(* Logix 5000 project; controller WWTP_SEC_CLX vendor 1 type 14 code 54 rev 17.2; software revision 17.00; part 12 of 13 *)
(* tags used below, declared in another part *)
   I_M403_Fault : ALIAS FOR Local:3:I.DATA.4;
   I_M403_Fault_IOFault : ALIAS FOR Local:3:I.Fault.4;
   I_M403_InAuto : ALIAS FOR Local:3:I.DATA.5;
   I_M403_InAuto_IOFault : ALIAS FOR Local:3:I.Fault.5;
   I_M403_RunFdbk : ALIAS FOR Local:3:I.DATA.3;
   I_M403_RunFdbk_IOFault : ALIAS FOR Local:3:I.Fault.3;
   I_SecTk01_InAuto : ALIAS FOR Local:2:I.DATA.4;
   I_SecTk01_InAuto_IOFault : ALIAS FOR Local:2:I.Fault.4;
   I_SecTk01_RAS_Flow : ALIAS FOR Local:5:I.CH0DATA;
   I_SecTk01_RAS_Flow_IOFault : ALIAS FOR Local:5:I.CH0Fault;
   I_SecTk01_RunFdbk : ALIAS FOR Local:2:I.DATA.3;
   I_SecTk01_RunFdbk_IOFault : ALIAS FOR Local:2:I.Fault.3;
   I_SecTk01_Torque : ALIAS FOR Local:2:I.DATA.5;
   I_SecTk01_Torque_IOFault : ALIAS FOR Local:2:I.Fault.5;
   O_M403_Out_Run : ALIAS FOR Local:4:O.DATA.6;   // M-402 Start/Stop
   O_SecTk01_Out_Run : ALIAS FOR Local:4:O.DATA.0;   // Secondary Tank #1 Start/Stop
   PLC_CommFail : U_CommFail;
   PLC_Device_ResetPB : BOOL;   // Site Wide Device Reset Push Button
   PLC_Heartbeat : U_Heartbeat;   // PLC Heartbeat
   PLC_Simulation : BOOL;   // Application running IN SIMULATION
   PLC_WallClock : U_WallClock;   // Wall Clock
   PRIM_FLOW_FIT302 : P_AIn;   // Primary Treatment Flow (FIT-302)
(* AerationTk02_Mixer01, continued *)

ROUTINE Main   (* ladder *)
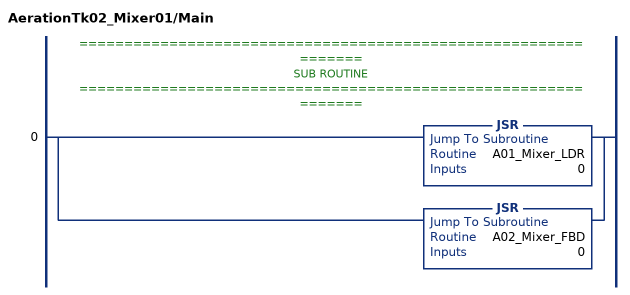
   // ===============================================================
   // SUB ROUTINE
   // ===============================================================
   0: [JSR(A01_Mixer_LDR,0) ,JSR(A02_Mixer_FBD,0) ];
END_ROUTINE
END_PROGRAM

PROGRAM AerationTk02_Mixer02   (* main routine Main *)
VAR
   Equip_Fault : ALIAS FOR I_M403_Fault;
   Equip_Fault_IOFault : ALIAS FOR I_M403_Fault_IOFault;
   Equip_GroupReset : ALIAS FOR PLC_Device_ResetPB;
   Equip_InAuto : ALIAS FOR I_M403_InAuto;
   Equip_InAuto_IOFault : ALIAS FOR I_M403_InAuto_IOFault;
   Equip_Intlk : ALIAS FOR M403_Intlk;
   Equip_IOFault : BOOL := 1;
   Equip_Motor : ALIAS FOR M403_Motor;
   Equip_Out_Run : ALIAS FOR O_M403_Out_Run;
   Equip_RunFdbk : ALIAS FOR I_M403_RunFdbk;
   Equip_RunFdbk_IOFault : ALIAS FOR I_M403_RunFdbk_IOFault;
   Wrk_Hand : BOOL;
   Wrk_ResetReqd : BOOL;
   Wrk_ResetRequired : BOOL;
END_VAR

ROUTINE A01_Mixer_LDR   (* ladder *)
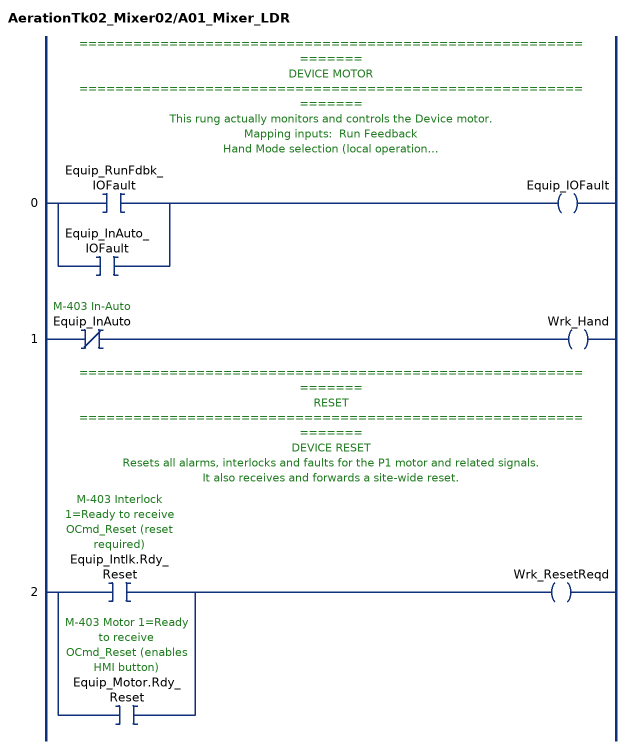
   // ===============================================================
   // DEVICE MOTOR
   // ===============================================================
   // This rung actually monitors and controls the Device motor.
   // Mapping inputs:  Run Feedback
   // Hand Mode selection (local operation)
   // Permissive OK
   // Protective’s OK,
   // I/O Fault signals
   // Pump Reset (above)
   // DEVICE
   // Output Mapping: Starter output
   0: [XIC(Equip_RunFdbk_IOFault) ,XIC(Equip_InAuto_IOFault) ]OTE(Equip_IOFault);
   1: XIO(Equip_InAuto)OTE(Wrk_Hand);
   // ===============================================================
   // RESET
   // ===============================================================
   // DEVICE RESET
   // Resets all alarms, interlocks and faults for the P1 motor and related signals.
   // It also receives and forwards a site-wide reset.
   2: [XIC(Equip_Intlk.Rdy_Reset) ,XIC(Equip_Motor.Rdy_Reset) ]OTE(Wrk_ResetReqd);
END_ROUTINE

ROUTINE A02_Mixer_FBD   (* function block diagram *)
   SHEET 1   // Motor
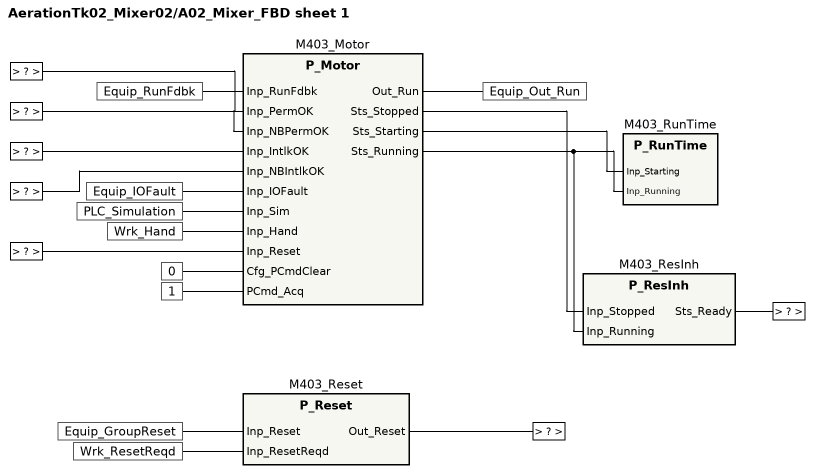
   M403_Reset : P_Reset(Inp_Reset := Equip_GroupReset, Inp_ResetReqd := Wrk_ResetReqd);
   WIRE(?) := M403_Reset.Out_Reset;
   M403_ResInh : P_ResInh(Inp_Stopped := M403_Motor.Sts_Stopped {feedback}, Inp_Running := M403_Motor.Sts_Running {feedback});
   WIRE(?) := M403_ResInh.Sts_Ready;
   M403_Motor : P_Motor(Inp_RunFdbk := Equip_RunFdbk, Inp_PermOK := WIRE(?), Inp_NBPermOK := WIRE(?), Inp_IntlkOK := WIRE(?), Inp_NBIntlkOK := WIRE(?), Inp_IOFault := Equip_IOFault, Inp_Sim := PLC_Simulation, Inp_Hand := Wrk_Hand, Inp_Reset := WIRE(?), Cfg_PCmdClear := 0, PCmd_Acq := 1);
   Equip_Out_Run := M403_Motor.Out_Run;
   M403_RunTime : P_RunTime(Inp_Starting := M403_Motor.Sts_Starting, Inp_Running := M403_Motor.Sts_Running);
   SHEET 2   // Permissives / Interlocks
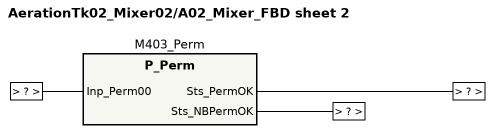
   M403_Perm : P_Perm(Inp_Perm00 := WIRE(?));
   WIRE(?) := M403_Perm.Sts_NBPermOK;
   WIRE(?) := M403_Perm.Sts_PermOK;
   SHEET 3   // Interlocks
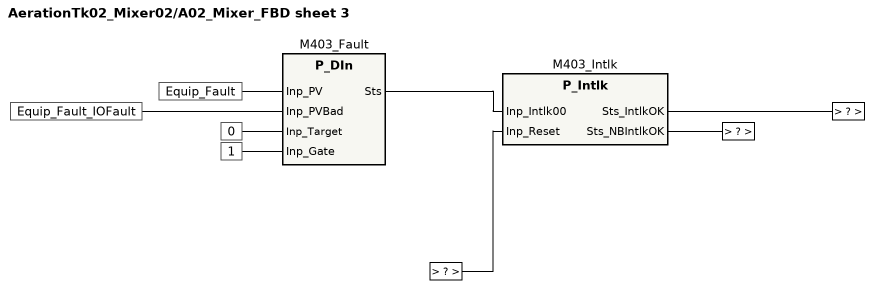
   M403_Fault : P_DIn(Inp_PV := Equip_Fault, Inp_PVBad := Equip_Fault_IOFault, Inp_Target := 0, Inp_Gate := 1);
   M403_Intlk : P_Intlk(Inp_Intlk00 := M403_Fault.Sts, Inp_Reset := WIRE(?));
   WIRE(?) := M403_Intlk.Sts_NBIntlkOK;
   WIRE(?) := M403_Intlk.Sts_IntlkOK;
END_ROUTINE

ROUTINE Main   (* ladder *)
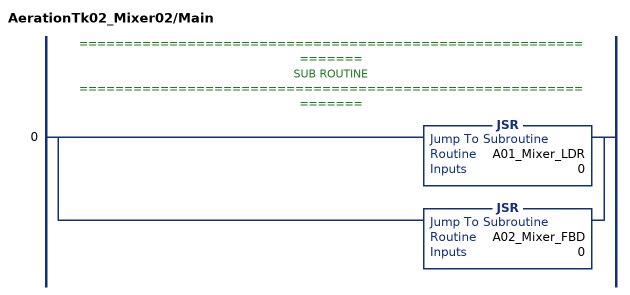
   // ===============================================================
   // SUB ROUTINE
   // ===============================================================
   0: [JSR(A01_Mixer_LDR,0) ,JSR(A02_Mixer_FBD,0) ];
END_ROUTINE
END_PROGRAM

PROGRAM MainProgram   (* main routine Main *)

ROUTINE A01_MiscDiscreteInputs   (* function block diagram *)
   SHEET 1
END_ROUTINE

ROUTINE A02_MiscAnalogInputs   (* function block diagram *)
   SHEET 1
END_ROUTINE

ROUTINE A03_MiscDiscreteOutputs   (* function block diagram *)
   SHEET 1
END_ROUTINE

ROUTINE A04_MiscAnalogOutputs   (* function block diagram *)
   SHEET 1
END_ROUTINE

ROUTINE Main   (* ladder *)
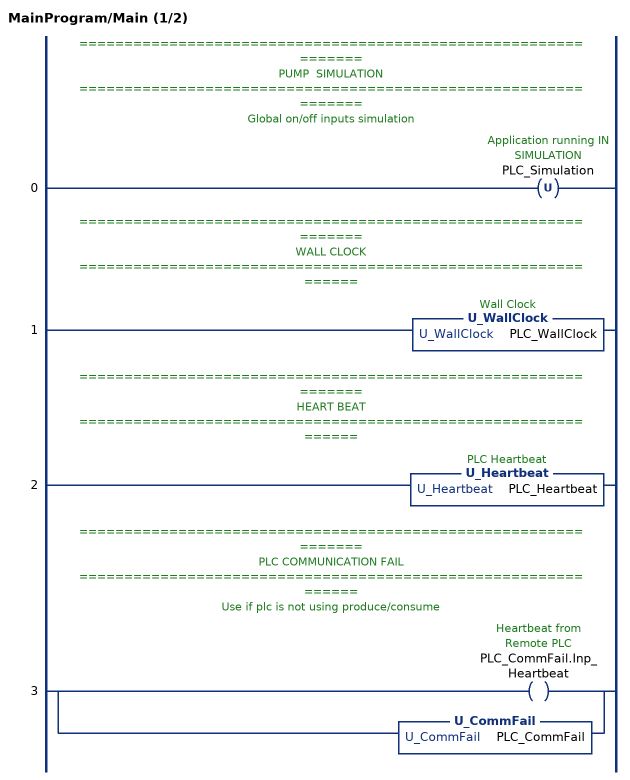
   // ===============================================================
   // PUMP  SIMULATION
   // ===============================================================
   // Global on/off inputs simulation
   0: OTU(PLC_Simulation);
   // ===============================================================
   // WALL CLOCK
   // ==============================================================
   1: U_WallClock(PLC_WallClock);
   // ===============================================================
   // HEART BEAT
   // ==============================================================
   2: U_Heartbeat(PLC_Heartbeat);
   // ===============================================================
   // PLC COMMUNICATION FAIL
   // ==============================================================
   // Use if plc is not using produce/consume
   3: [OTE(PLC_CommFail.Inp_Heartbeat) ,U_CommFail(PLC_CommFail) ];
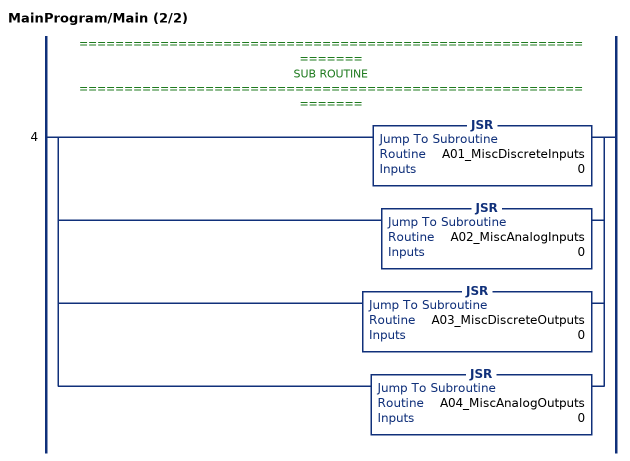
   // ===============================================================
   // SUB ROUTINE
   // ===============================================================
   4: [JSR(A01_MiscDiscreteInputs,0) ,JSR(A02_MiscAnalogInputs,0) ,JSR(A03_MiscDiscreteOutputs,0) ,JSR(A04_MiscAnalogOutputs,0) ];
END_ROUTINE
END_PROGRAM

PROGRAM SecTank01_Drive   (* main routine Main *)
VAR
   Equip_GroupReset : ALIAS FOR PLC_Device_ResetPB;
   Equip_InAuto : ALIAS FOR I_SecTk01_InAuto;
   Equip_InAuto_IOFault : ALIAS FOR I_SecTk01_InAuto_IOFault;
   Equip_Intlk : ALIAS FOR SecTk01_Intlk;
   Equip_IOFault : BOOL;
   Equip_Motor : ALIAS FOR SecTk01_Motor;
   Equip_Out_Run : ALIAS FOR O_SecTk01_Out_Run;
   Equip_RunFdbk : ALIAS FOR I_SecTk01_RunFdbk;
   Equip_RunFdbk_IOFault : ALIAS FOR I_SecTk01_RunFdbk_IOFault;
   Equip_Torque : ALIAS FOR I_SecTk01_Torque;
   Equip_Torque_IOFault : ALIAS FOR I_SecTk01_Torque_IOFault;
   Wrk_Hand : BOOL;
   Wrk_ResetReqd : BOOL := 1;
   Wrk_ResetRequired : BOOL;
END_VAR

ROUTINE A01_Drive_LDR   (* ladder *)
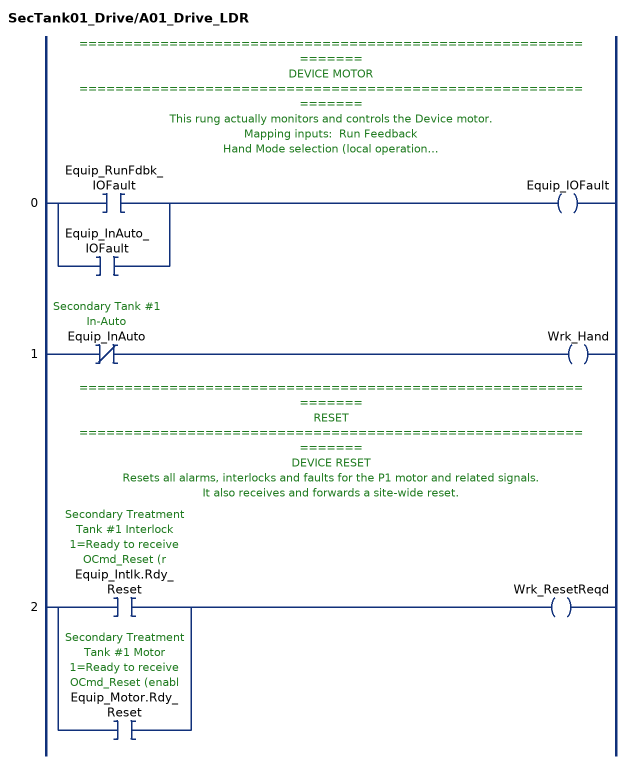
   // ===============================================================
   // DEVICE MOTOR
   // ===============================================================
   // This rung actually monitors and controls the Device motor.
   // Mapping inputs:  Run Feedback
   // Hand Mode selection (local operation)
   // Permissive OK
   // Protective’s OK,
   // I/O Fault signals
   // Pump Reset (above)
   // DEVICE
   // Output Mapping: Starter output
   0: [XIC(Equip_RunFdbk_IOFault) ,XIC(Equip_InAuto_IOFault) ]OTE(Equip_IOFault);
   1: XIO(Equip_InAuto)OTE(Wrk_Hand);
   // ===============================================================
   // RESET
   // ===============================================================
   // DEVICE RESET
   // Resets all alarms, interlocks and faults for the P1 motor and related signals.
   // It also receives and forwards a site-wide reset.
   2: [XIC(Equip_Intlk.Rdy_Reset) ,XIC(Equip_Motor.Rdy_Reset) ]OTE(Wrk_ResetReqd);
END_ROUTINE

ROUTINE A02_Drive_FBD   (* function block diagram *)
   SHEET 1   // Motor
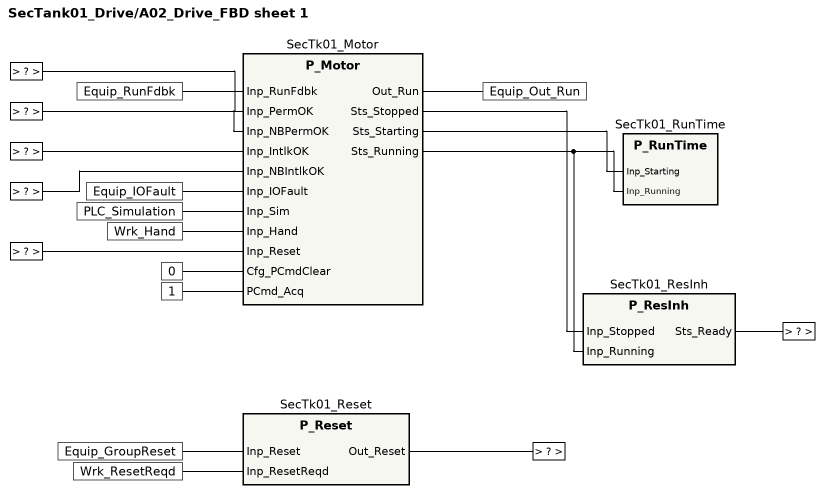
   SecTk01_Reset : P_Reset(Inp_Reset := Equip_GroupReset, Inp_ResetReqd := Wrk_ResetReqd);
   WIRE(?) := SecTk01_Reset.Out_Reset;
   SecTk01_ResInh : P_ResInh(Inp_Stopped := SecTk01_Motor.Sts_Stopped {feedback}, Inp_Running := SecTk01_Motor.Sts_Running {feedback});
   WIRE(?) := SecTk01_ResInh.Sts_Ready;
   SecTk01_Motor : P_Motor(Inp_RunFdbk := Equip_RunFdbk, Inp_PermOK := WIRE(?), Inp_NBPermOK := WIRE(?), Inp_IntlkOK := WIRE(?), Inp_NBIntlkOK := WIRE(?), Inp_IOFault := Equip_IOFault, Inp_Sim := PLC_Simulation, Inp_Hand := Wrk_Hand, Inp_Reset := WIRE(?), Cfg_PCmdClear := 0, PCmd_Acq := 1);
   Equip_Out_Run := SecTk01_Motor.Out_Run;
   SecTk01_RunTime : P_RunTime(Inp_Starting := SecTk01_Motor.Sts_Starting, Inp_Running := SecTk01_Motor.Sts_Running);
   SHEET 2   // Permissives
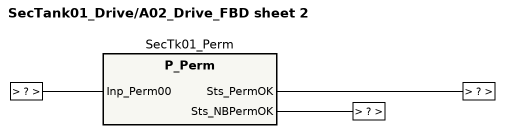
   SecTk01_Perm : P_Perm(Inp_Perm00 := WIRE(?));
   WIRE(?) := SecTk01_Perm.Sts_NBPermOK;
   WIRE(?) := SecTk01_Perm.Sts_PermOK;
   SHEET 3   // Interlocks
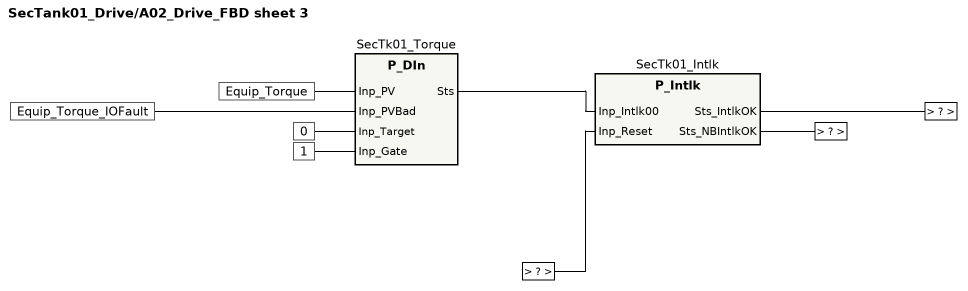
   SecTk01_Torque : P_DIn(Inp_PV := Equip_Torque, Inp_PVBad := Equip_Torque_IOFault, Inp_Target := 0, Inp_Gate := 1);
   SecTk01_Intlk : P_Intlk(Inp_Intlk00 := SecTk01_Torque.Sts, Inp_Reset := WIRE(?));
   WIRE(?) := SecTk01_Intlk.Sts_NBIntlkOK;
   WIRE(?) := SecTk01_Intlk.Sts_IntlkOK;
END_ROUTINE

ROUTINE Main   (* ladder *)
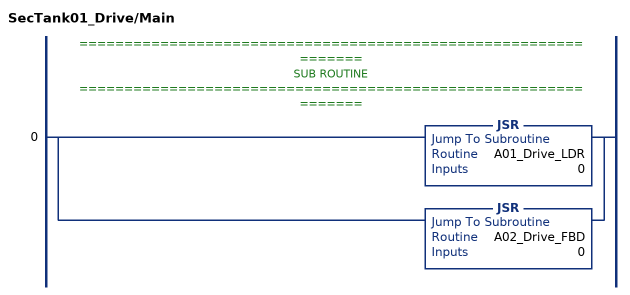
   // ===============================================================
   // SUB ROUTINE
   // ===============================================================
   0: [JSR(A01_Drive_LDR,0) ,JSR(A02_Drive_FBD,0) ];
END_ROUTINE
END_PROGRAM

PROGRAM SecTank01_RAS_Pump   (* main routine Main *)
VAR
   Equip_GroupReset : ALIAS FOR PLC_Device_ResetPB;
   Equip_Intlk : ALIAS FOR RAS_P401_Intlk;
   Equip_IOFault : BOOL;
   Equip_Motor : ALIAS FOR RAS_P401_VSD;
   Equip_RAS_Flow : ALIAS FOR I_SecTk01_RAS_Flow;
   Equip_RAS_Flow_IOFault : ALIAS FOR I_SecTk01_RAS_Flow_IOFault;
   Equip_RatioFlow : ALIAS FOR PRIM_FLOW_FIT302;
   Equip_VFD_I : ALIAS FOR WWTP_RAS_P401:I;
   Equip_VFD_O : ALIAS FOR WWTP_RAS_P401:O;
   Wrk_Hand : BOOL;
   Wrk_ResetReqd : BOOL;
   Wrk_ResetRequired : BOOL;
END_VAR

ROUTINE A01_Pump_LDR   (* ladder *)
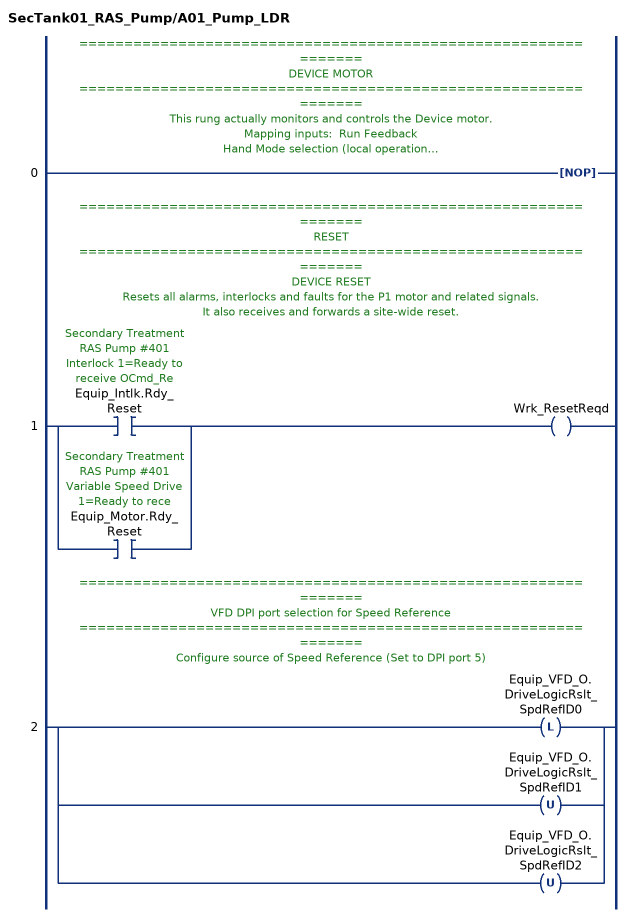
   // ===============================================================
   // DEVICE MOTOR
   // ===============================================================
   // This rung actually monitors and controls the Device motor.
   // Mapping inputs:  Run Feedback
   // Hand Mode selection (local operation)
   // Permissive OK
   // Protective’s OK,
   // I/O Fault signals
   // Pump Reset (above)
   // DEVICE
   // Output Mapping: Starter output
   0: NOP();
   // ===============================================================
   // RESET
   // ===============================================================
   // DEVICE RESET
   // Resets all alarms, interlocks and faults for the P1 motor and related signals.
   // It also receives and forwards a site-wide reset.
   1: [XIC(Equip_Intlk.Rdy_Reset) ,XIC(Equip_Motor.Rdy_Reset) ]OTE(Wrk_ResetReqd);
   // ===============================================================
   // VFD DPI port selection for Speed Reference
   // ===============================================================
   // Configure source of Speed Reference (Set to DPI port 5)
   2: [OTL(Equip_VFD_O.DriveLogicRslt_SpdRefID0) ,OTU(Equip_VFD_O.DriveLogicRslt_SpdRefID1) ,OTU(Equip_VFD_O.DriveLogicRslt_SpdRefID2) ];
END_ROUTINE

ROUTINE A02_Pump_FBD   (* function block diagram *)
   SHEET 1   // Motor
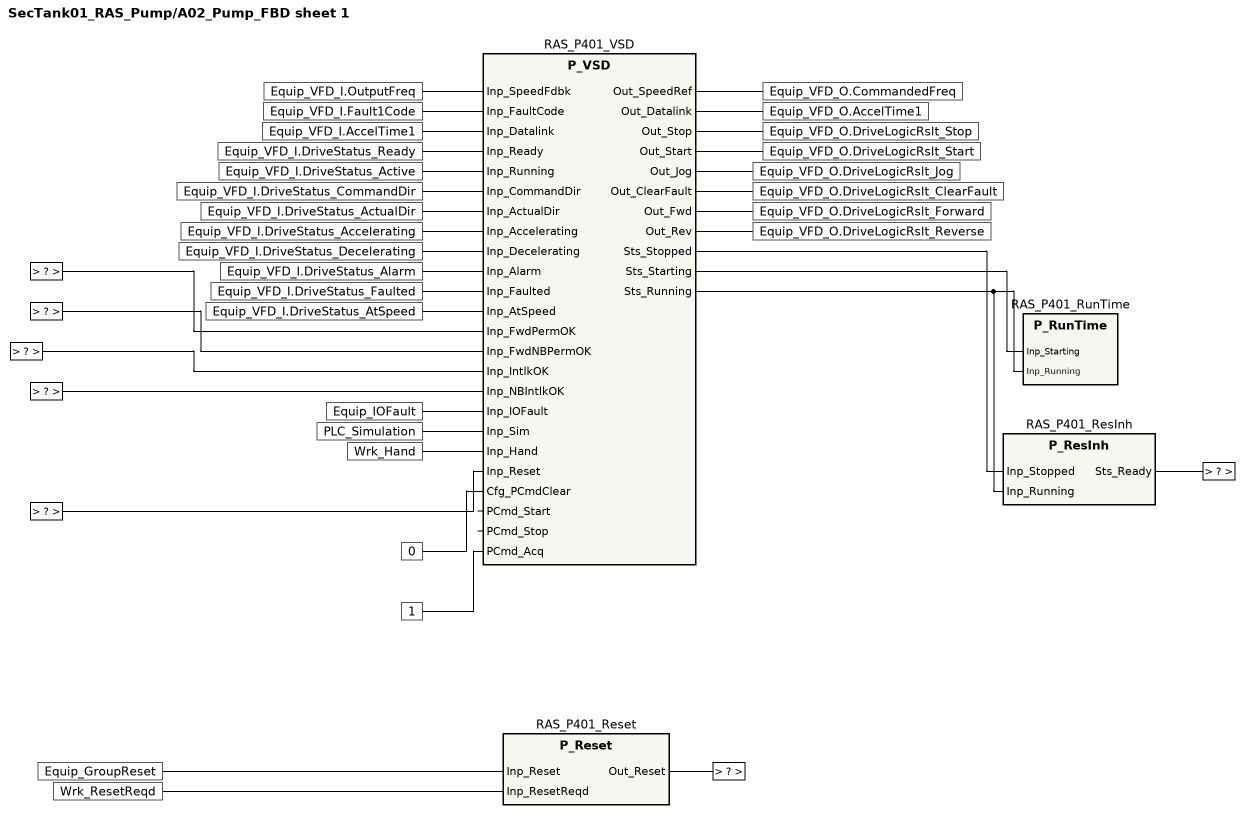
   RAS_P401_Reset : P_Reset(Inp_Reset := Equip_GroupReset, Inp_ResetReqd := Wrk_ResetReqd);
   WIRE(?) := RAS_P401_Reset.Out_Reset;
   RAS_P401_ResInh : P_ResInh(Inp_Stopped := RAS_P401_VSD.Sts_Stopped {feedback}, Inp_Running := RAS_P401_VSD.Sts_Running {feedback});
   WIRE(?) := RAS_P401_ResInh.Sts_Ready;
   RAS_P401_VSD : P_VSD(Inp_SpeedFdbk := Equip_VFD_I.OutputFreq, Inp_FaultCode := Equip_VFD_I.Fault1Code, Inp_Datalink := Equip_VFD_I.AccelTime1, Inp_Ready := Equip_VFD_I.DriveStatus_Ready, Inp_Running := Equip_VFD_I.DriveStatus_Active, Inp_CommandDir := Equip_VFD_I.DriveStatus_CommandDir, Inp_ActualDir := Equip_VFD_I.DriveStatus_ActualDir, Inp_Accelerating := Equip_VFD_I.DriveStatus_Accelerating, Inp_Decelerating := Equip_VFD_I.DriveStatus_Decelerating, Inp_Alarm := Equip_VFD_I.DriveStatus_Alarm, Inp_Faulted := Equip_VFD_I.DriveStatus_Faulted, Inp_AtSpeed := Equip_VFD_I.DriveStatus_AtSpeed, Inp_FwdPermOK := WIRE(?), Inp_FwdNBPermOK := WIRE(?), Inp_IntlkOK := WIRE(?), Inp_NBIntlkOK := WIRE(?), Inp_IOFault := Equip_IOFault, Inp_Sim := PLC_Simulation, Inp_Hand := Wrk_Hand, Inp_Reset := WIRE(?), Cfg_PCmdClear := 0, PCmd_Acq := 1);   // unwired pins: PCmd_Start PCmd_Stop
   Equip_VFD_O.DriveLogicRslt_Jog := RAS_P401_VSD.Out_Jog;
   Equip_VFD_O.DriveLogicRslt_ClearFault := RAS_P401_VSD.Out_ClearFault;
   Equip_VFD_O.DriveLogicRslt_Forward := RAS_P401_VSD.Out_Fwd;
   Equip_VFD_O.DriveLogicRslt_Reverse := RAS_P401_VSD.Out_Rev;
   Equip_VFD_O.CommandedFreq := RAS_P401_VSD.Out_SpeedRef;
   Equip_VFD_O.AccelTime1 := RAS_P401_VSD.Out_Datalink;
   Equip_VFD_O.DriveLogicRslt_Stop := RAS_P401_VSD.Out_Stop;
   Equip_VFD_O.DriveLogicRslt_Start := RAS_P401_VSD.Out_Start;
   RAS_P401_RunTime : P_RunTime(Inp_Starting := RAS_P401_VSD.Sts_Starting, Inp_Running := RAS_P401_VSD.Sts_Running);
   SHEET 2   // Permissives
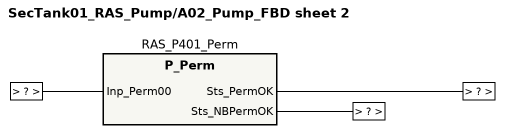
   RAS_P401_Perm : P_Perm(Inp_Perm00 := WIRE(?));
   WIRE(?) := RAS_P401_Perm.Sts_NBPermOK;
   WIRE(?) := RAS_P401_Perm.Sts_PermOK;
   SHEET 3   // Interlocks
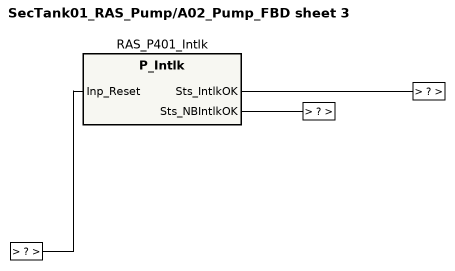
   RAS_P401_Intlk : P_Intlk(Inp_Reset := WIRE(?));
   WIRE(?) := RAS_P401_Intlk.Sts_NBIntlkOK;
   WIRE(?) := RAS_P401_Intlk.Sts_IntlkOK;
END_ROUTINE

ROUTINE A04_PumpDischargeFlow   (* function block diagram *)
   SHEET 1
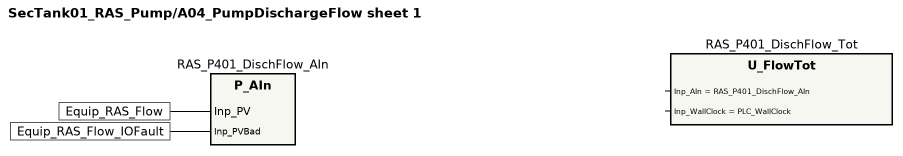
   RAS_P401_DischFlow_AIn : P_AIn(Inp_PV := Equip_RAS_Flow, Inp_PVBad := Equip_RAS_Flow_IOFault);
   RAS_P401_DischFlow_Tot : U_FlowTot(Inp_AIn := RAS_P401_DischFlow_AIn, Inp_WallClock := PLC_WallClock);
END_ROUTINE
